  MoveL 690 to (-312.65, 5.37, -312.58) mm, rotated rx -179.15 ry 0 rz -30.08 deg; joints [-2.468, -65.05, 119.495, -183.449, 54.303, 242.138]
  MoveL 691 to (-312.62, 5.43, -312.23) mm, rotated rx -179.15 ry 0 rz -30.08 deg; joints [-2.467, -65.071, 119.523, -183.448, 54.309, 242.137]
  MoveL 692 to (-312.59, 5.47, -311.88) mm, rotated rx -179.15 ry 0 rz -30.08 deg; joints [-2.466, -65.091, 119.551, -183.447, 54.317, 242.136]
  MoveL 693 to (-312.58, 5.49, -311.54) mm, rotated rx -179.15 ry 0 rz -30.08 deg; joints [-2.466, -65.11, 119.579, -183.447, 54.326, 242.135]
  MoveL 694 to (-312.58, 5.49, -311.19) mm, rotated rx -179.15 ry 0 rz -30.08 deg; joints [-2.467, -65.129, 119.607, -183.447, 54.336, 242.135]
  MoveL 695 to (-312.58, 5.49, -5.24) mm, rotated rx -179.15 ry 0 rz -30.08 deg; joints [-3.196, -81.654, 142.775, -184.036, 60.99, 242.081]
  MoveL 696 to (-312.58, 5.49, -2.45) mm, rotated rx -179.15 ry 0 rz -30.08 deg; joints [-3.205, -81.818, 142.973, -184.044, 61.024, 242.083]
  MoveL 697 to (-312.59, 5.47, -2.1) mm, rotated rx -179.15 ry 0 rz -30.08 deg; joints [-3.206, -81.837, 142.998, -184.046, 61.03, 242.083]
  MoveL 698 to (-312.62, 5.43, -1.75) mm, rotated rx -179.15 ry 0 rz -30.08 deg; joints [-3.209, -81.854, 143.023, -184.049, 61.038, 242.084]
  MoveL 699 to (-312.65, 5.37, -1.4) mm, rotated rx -179.15 ry 0 rz -30.08 deg; joints [-3.212, -81.871, 143.049, -184.052, 61.048, 242.085]
  MoveL 700 to (-312.69, 5.3, -1.05) mm, rotated rx -179.15 ry 0 rz -30.08 deg; joints [-3.215, -81.886, 143.075, -184.055, 61.059, 242.086]
  MoveL 701 to (-312.75, 5.2, -0.7) mm, rotated rx -179.15 ry 0 rz -30.08 deg; joints [-3.22, -81.9, 143.102, -184.06, 61.072, 242.087]
  MoveL 702 to (-312.81, 5.09, -0.35) mm, rotated rx -179.15 ry 0 rz -30.08 deg; joints [-3.224, -81.912, 143.129, -184.065, 61.087, 242.089]
  MoveL 703 to (-312.89, 4.96, 0) mm, rotated rx -179.15 ry 0 rz -30.08 deg; joints [-3.23, -81.923, 143.156, -184.07, 61.103, 242.09]
  MoveL 704 to (-312.98, 4.8, 0.35) mm, rotated rx -179.15 ry 0 rz -30.08 deg; joints [-3.236, -81.932, 143.184, -184.077, 61.122, 242.092]
  MoveL 705 to (-313.06, 4.67, 0.61) mm, rotated rx -179.15 ry 0 rz -30.08 deg; joints [-3.242, -81.938, 143.205, -184.082, 61.138, 242.094]
  MoveL 706 to (-313.14, 4.52, 0.87) mm, rotated rx -179.15 ry 0 rz -30.08 deg; joints [-3.247, -81.942, 143.227, -184.088, 61.155, 242.096]
  MoveL 707 to (-313.28, 4.28, 1.23) mm, rotated rx -179.15 ry 0 rz -30.08 deg; joints [-3.256, -81.946, 143.257, -184.097, 61.181, 242.099]
  MoveL 708 to (-313.44, 4.01, 1.6) mm, rotated rx -179.15 ry 0 rz -30.08 deg; joints [-3.267, -81.948, 143.288, -184.108, 61.211, 242.102]
  MoveL 709 to (-313.54, 3.84, 1.8) mm, rotated rx -179.15 ry 0 rz -30.08 deg; joints [-3.273, -81.947, 143.306, -184.115, 61.23, 242.104]
  MoveL 710 to (-313.64, 3.66, 1.99) mm, rotated rx -179.15 ry 0 rz -30.08 deg; joints [-3.279, -81.945, 143.323, -184.121, 61.249, 242.106]
  MoveL 711 to (-313.84, 3.31, 2.32) mm, rotated rx -179.15 ry 0 rz -30.08 deg; joints [-3.292, -81.939, 143.354, -184.134, 61.286, 242.11]
  MoveL 712 to (-314.02, 3.01, 2.57) mm, rotated rx -179.15 ry 0 rz -30.08 deg; joints [-3.303, -81.932, 143.377, -184.145, 61.317, 242.113]
  MoveL 713 to (-314.19, 2.71, 2.78) mm, rotated rx -179.15 ry 0 rz -30.08 deg; joints [-3.314, -81.922, 143.398, -184.156, 61.348, 242.116]
  MoveL 714 to (-314.37, 2.41, 2.96) mm, rotated rx -179.15 ry 0 rz -30.08 deg; joints [-3.325, -81.91, 143.417, -184.167, 61.379, 242.12]
  MoveL 715 to (-314.54, 2.1, 3.12) mm, rotated rx -179.15 ry 0 rz -30.08 deg; joints [-3.335, -81.898, 143.435, -184.178, 61.41, 242.123]
  MoveL 716 to (-314.57, 2.06, 3.14) mm, rotated rx -179.15 ry 0 rz -30.08 deg; joints [-3.337, -81.896, 143.437, -184.18, 61.414, 242.123]
  MoveL 717 to (-314.74, 1.76, 3.27) mm, rotated rx -179.15 ry 0 rz -30.08 deg; joints [-3.347, -81.881, 143.452, -184.19, 61.443, 242.126]
  MoveL 718 to (-314.91, 1.47, 3.37) mm, rotated rx -179.15 ry 0 rz -30.08 deg; joints [-3.357, -81.866, 143.465, -184.201, 61.473, 242.129]
  MoveL 719 to (-315.08, 1.17, 3.46) mm, rotated rx -179.15 ry 0 rz -30.08 deg; joints [-3.367, -81.849, 143.477, -184.211, 61.502, 242.133]
  MoveL 720 to (-315.25, 0.88, 3.52) mm, rotated rx -179.15 ry 0 rz -30.08 deg; joints [-3.377, -81.831, 143.487, -184.222, 61.531, 242.136]
  MoveL 721 to (-315.43, 0.58, 3.57) mm, rotated rx -179.15 ry 0 rz -30.08 deg; joints [-3.387, -81.811, 143.497, -184.232, 61.559, 242.139]
  MoveL 722 to (-315.6, 0.28, 3.6) mm, rotated rx -179.15 ry 0 rz -30.08 deg; joints [-3.397, -81.791, 143.504, -184.242, 61.588, 242.142]
  MoveL 723 to (-315.94, -0.31, 3.61) mm, rotated rx -179.15 ry 0 rz -30.08 deg; joints [-3.417, -81.748, 143.517, -184.262, 61.644, 242.148]
  MoveL 724 to (-316.64, -1.52, 3.61) mm, rotated rx -179.15 ry 0 rz -30.08 deg; joints [-3.458, -81.658, 143.54, -184.304, 61.758, 242.16]
  MoveL 725 to (-316.99, -2.12, 3.58) mm, rotated rx -179.15 ry 0 rz -30.08 deg; joints [-3.478, -81.612, 143.551, -184.324, 61.815, 242.165]
  MoveL 726 to (-317.34, -2.72, 3.49) mm, rotated rx -179.15 ry 0 rz -30.08 deg; joints [-3.498, -81.562, 143.556, -184.344, 61.871, 242.171]
  MoveL 727 to (-321.53, -9.97, 2.16) mm, rotated rx -179.15 ry 0 rz -30.08 deg; joints [-3.734, -80.943, 143.599, -184.585, 62.54, 242.237]
  MoveL 728 to (-322.93, -12.38, 1.71) mm, rotated rx -179.15 ry 0 rz -30.08 deg; joints [-3.813, -80.735, 143.611, -184.664, 62.762, 242.257]
  MoveL 729 to (-323.1, -12.68, 1.62) mm, rotated rx -179.15 ry 0 rz -30.08 deg; joints [-3.823, -80.707, 143.61, -184.674, 62.788, 242.26]
  MoveL 730 to (-323.28, -12.97, 1.52) mm, rotated rx -179.15 ry 0 rz -30.08 deg; joints [-3.832, -80.679, 143.608, -184.683, 62.815, 242.262]
  MoveL 731 to (-323.45, -13.27, 1.39) mm, rotated rx -179.15 ry 0 rz -30.08 deg; joints [-3.841, -80.649, 143.604, -184.693, 62.841, 242.265]
  MoveL 732 to (-323.62, -13.56, 1.24) mm, rotated rx -179.15 ry 0 rz -30.08 deg; joints [-3.851, -80.618, 143.598, -184.702, 62.867, 242.267]
  MoveL 733 to (-323.79, -13.86, 1.06) mm, rotated rx -179.15 ry 0 rz -30.08 deg; joints [-3.86, -80.586, 143.591, -184.711, 62.892, 242.269]
  MoveL 734 to (-323.96, -14.15, 0.85) mm, rotated rx -179.15 ry 0 rz -30.08 deg; joints [-3.869, -80.552, 143.582, -184.72, 62.917, 242.272]
  MoveL 735 to (-324.13, -14.45, 0.62) mm, rotated rx -179.15 ry 0 rz -30.08 deg; joints [-3.878, -80.516, 143.57, -184.729, 62.942, 242.274]
  MoveL 736 to (-324.3, -14.74, 0.35) mm, rotated rx -179.15 ry 0 rz -30.08 deg; joints [-3.887, -80.478, 143.556, -184.738, 62.966, 242.276]
  MoveL 737 to (-324.33, -14.8, 0.3) mm, rotated rx -179.15 ry 0 rz -30.08 deg; joints [-3.888, -80.472, 143.554, -184.74, 62.97, 242.277]
  MoveC 738 to (-325.22, -16.33, 0.41) mm, rotated rx -179.15 ry 0 rz -30.08 deg; joints [-3.94, -80.362, 143.589, -184.791, 63.116, 242.289] to (-325.18, -16.27, 2.18) mm, rotated rx -179.15 ry 0 rz -30.08 deg; joints [-3.944, -80.467, 143.714, -184.796, 63.136, 242.29]
  MoveL 739 to (-325.18, -16.27, 2.18) mm, rotated rx -179.15 ry 0 rz -30.08 deg; joints [-3.944, -80.467, 143.714, -184.796, 63.136, 242.29]
  MoveL 740 to (-324.74, -15.51, 3.02) mm, rotated rx -179.15 ry 0 rz -30.08 deg; joints [-3.922, -80.573, 143.76, -184.774, 63.076, 242.284]
  Set speed (50.0 mm/s)
  MoveL 741 to (-322.97, -16.53, 3.02) mm, rotated rx -179.15 ry 0 rz -30.08 deg; joints [-3.82, -80.504, 143.789, -184.655, 63.169, 242.224]
  MoveL 742 to (-321.44, -16.41, 2.09) mm, rotated rx -179.15 ry 0 rz -30.08 deg; joints [-3.727, -80.466, 143.728, -184.552, 63.143, 242.179]
  Set speed (100.0 mm/s)
  MoveC 743 to (-321.26, -16.11, 1.18) mm, rotated rx -179.15 ry 0 rz -30.08 deg; joints [-3.714, -80.437, 143.658, -184.539, 63.101, 242.176] to (-321.46, -16.46, 0.3) mm, rotated rx -179.15 ry 0 rz -30.08 deg; joints [-3.722, -80.361, 143.601, -184.547, 63.121, 242.179]
  MoveL 744 to (-321.46, -16.46, 0.3) mm, rotated rx -179.15 ry 0 rz -30.08 deg; joints [-3.722, -80.361, 143.601, -184.547, 63.121, 242.179]
  MoveL 745 to (-321.65, -16.77, -0.05) mm, rotated rx -179.15 ry 0 rz -30.08 deg; joints [-3.732, -80.317, 143.582, -184.557, 63.146, 242.181]
  MoveL 746 to (-321.8, -17.04, -0.39) mm, rotated rx -179.15 ry 0 rz -30.08 deg; joints [-3.739, -80.277, 143.562, -184.565, 63.166, 242.183]
  MoveL 747 to (-321.94, -17.28, -0.73) mm, rotated rx -179.15 ry 0 rz -30.08 deg; joints [-3.746, -80.24, 143.542, -184.571, 63.183, 242.185]
  MoveL 748 to (-322.05, -17.48, -1.07) mm, rotated rx -179.15 ry 0 rz -30.08 deg; joints [-3.751, -80.205, 143.521, -184.577, 63.198, 242.186]
  MoveL 749 to (-322.16, -17.66, -1.42) mm, rotated rx -179.15 ry 0 rz -30.08 deg; joints [-3.756, -80.173, 143.5, -184.581, 63.209, 242.188]
  MoveL 750 to (-322.25, -17.81, -1.76) mm, rotated rx -179.15 ry 0 rz -30.08 deg; joints [-3.76, -80.142, 143.478, -184.585, 63.218, 242.189]
  MoveL 751 to (-322.32, -17.94, -2.1) mm, rotated rx -179.15 ry 0 rz -30.08 deg; joints [-3.763, -80.112, 143.456, -184.589, 63.226, 242.19]
  MoveL 752 to (-322.38, -18.05, -2.45) mm, rotated rx -179.15 ry 0 rz -30.08 deg; joints [-3.765, -80.085, 143.433, -184.591, 63.231, 242.19]
  MoveL 753 to (-322.44, -18.14, -2.8) mm, rotated rx -179.15 ry 0 rz -30.08 deg; joints [-3.767, -80.058, 143.41, -184.593, 63.235, 242.191]
  MoveL 754 to (-322.48, -18.22, -3.14) mm, rotated rx -179.15 ry 0 rz -30.08 deg; joints [-3.768, -80.033, 143.386, -184.594, 63.236, 242.191]
  MoveL 755 to (-322.51, -18.27, -3.49) mm, rotated rx -179.15 ry 0 rz -30.08 deg; joints [-3.769, -80.009, 143.362, -184.595, 63.236, 242.192]
  MoveL 756 to (-322.54, -18.31, -3.84) mm, rotated rx -179.15 ry 0 rz -30.08 deg; joints [-3.769, -79.986, 143.338, -184.595, 63.235, 242.192]
  MoveL 757 to (-322.55, -18.33, -4.19) mm, rotated rx -179.15 ry 0 rz -30.08 deg; joints [-3.768, -79.964, 143.314, -184.594, 63.232, 242.192]
  MoveL 758 to (-322.55, -18.34, -4.54) mm, rotated rx -179.15 ry 0 rz -30.08 deg; joints [-3.767, -79.944, 143.289, -184.593, 63.227, 242.192]
  MoveL 759 to (-322.55, -18.34, -311.19) mm, rotated rx -179.15 ry 0 rz -30.08 deg; joints [-2.902, -63.912, 119.964, -183.907, 55.922, 242.314]
  MoveL 760 to (-322.55, -18.33, -311.54) mm, rotated rx -179.15 ry 0 rz -30.08 deg; joints [-2.901, -63.895, 119.935, -183.906, 55.911, 242.314]
  MoveL 761 to (-322.54, -18.31, -311.88) mm, rotated rx -179.15 ry 0 rz -30.08 deg; joints [-2.9, -63.878, 119.906, -183.905, 55.898, 242.314]
  MoveL 762 to (-322.51, -18.27, -312.23) mm, rotated rx -179.15 ry 0 rz -30.08 deg; joints [-2.898, -63.863, 119.877, -183.904, 55.885, 242.314]
  MoveL 763 to (-322.48, -18.22, -312.58) mm, rotated rx -179.15 ry 0 rz -30.08 deg; joints [-2.896, -63.848, 119.848, -183.902, 55.87, 242.314]
  MoveL 764 to (-322.44, -18.14, -312.93) mm, rotated rx -179.15 ry 0 rz -30.08 deg; joints [-2.894, -63.834, 119.818, -183.899, 55.854, 242.313]
  MoveL 765 to (-322.38, -18.05, -313.28) mm, rotated rx -179.15 ry 0 rz -30.08 deg; joints [-2.89, -63.821, 119.789, -183.896, 55.837, 242.312]
  MoveL 766 to (-322.32, -17.93, -313.63) mm, rotated rx -179.15 ry 0 rz -30.08 deg; joints [-2.887, -63.81, 119.759, -183.893, 55.819, 242.311]
  MoveL 767 to (-322.24, -17.8, -313.98) mm, rotated rx -179.15 ry 0 rz -30.08 deg; joints [-2.883, -63.799, 119.728, -183.889, 55.799, 242.31]
  MoveL 768 to (-322.15, -17.64, -314.33) mm, rotated rx -179.15 ry 0 rz -30.08 deg; joints [-2.878, -63.789, 119.698, -183.884, 55.778, 242.309]
  MoveL 769 to (-322.05, -17.46, -314.68) mm, rotated rx -179.15 ry 0 rz -30.08 deg; joints [-2.873, -63.781, 119.667, -183.879, 55.755, 242.307]
  MoveL 770 to (-321.92, -17.25, -315.03) mm, rotated rx -179.15 ry 0 rz -30.08 deg; joints [-2.867, -63.774, 119.635, -183.873, 55.73, 242.305]
  MoveL 771 to (-321.78, -17.01, -315.38) mm, rotated rx -179.15 ry 0 rz -30.08 deg; joints [-2.86, -63.769, 119.603, -183.866, 55.703, 242.303]
  MoveL 772 to (-321.63, -16.75, -315.7) mm, rotated rx -179.15 ry 0 rz -30.08 deg; joints [-2.853, -63.766, 119.574, -183.858, 55.676, 242.3]
  MoveL 773 to (-321.46, -16.46, -316.02) mm, rotated rx -179.15 ry 0 rz -30.08 deg; joints [-2.844, -63.765, 119.543, -183.85, 55.647, 242.297]
  MoveL 774 to (-321.29, -16.16, -316.3) mm, rotated rx -179.15 ry 0 rz -30.08 deg; joints [-2.836, -63.767, 119.516, -183.841, 55.618, 242.293]
  MoveL 775 to (-321.11, -15.85, -316.55) mm, rotated rx -179.15 ry 0 rz -30.08 deg; joints [-2.828, -63.77, 119.492, -183.832, 55.591, 242.29]
  MoveL 776 to (-320.94, -15.55, -316.76) mm, rotated rx -179.15 ry 0 rz -30.08 deg; joints [-2.82, -63.775, 119.471, -183.824, 55.564, 242.287]
  MoveL 777 to (-320.76, -15.25, -316.94) mm, rotated rx -179.15 ry 0 rz -30.08 deg; joints [-2.812, -63.781, 119.452, -183.815, 55.538, 242.283]
  MoveL 778 to (-320.59, -14.95, -317.1) mm, rotated rx -179.15 ry 0 rz -30.08 deg; joints [-2.804, -63.789, 119.435, -183.807, 55.514, 242.28]
  MoveL 779 to (-320.41, -14.65, -317.23) mm, rotated rx -179.15 ry 0 rz -30.08 deg; joints [-2.796, -63.798, 119.42, -183.798, 55.489, 242.276]
  MoveL 780 to (-320.24, -14.35, -317.34) mm, rotated rx -179.15 ry 0 rz -30.08 deg; joints [-2.788, -63.808, 119.407, -183.79, 55.466, 242.273]
  MoveL 781 to (-320.06, -14.04, -317.43) mm, rotated rx -179.15 ry 0 rz -30.08 deg; joints [-2.781, -63.819, 119.395, -183.781, 55.443, 242.269]
  MoveL 782 to (-319.89, -13.74, -317.5) mm, rotated rx -179.15 ry 0 rz -30.08 deg; joints [-2.773, -63.831, 119.386, -183.773, 55.421, 242.266]
  MoveL 783 to (-319.71, -13.44, -317.55) mm, rotated rx -179.15 ry 0 rz -30.08 deg; joints [-2.765, -63.844, 119.378, -183.765, 55.4, 242.262]
  MoveL 784 to (-319.54, -13.14, -317.58) mm, rotated rx -179.15 ry 0 rz -30.08 deg; joints [-2.758, -63.858, 119.371, -183.756, 55.379, 242.259]
  MoveL 785 to (-319.37, -12.84, -317.59) mm, rotated rx -179.15 ry 0 rz -30.08 deg; joints [-2.75, -63.873, 119.366, -183.748, 55.359, 242.255]
  MoveL 786 to (-312.02, -0.16, -317.59) mm, rotated rx -179.15 ry 0 rz -30.08 deg; joints [-2.43, -64.521, 119.184, -183.394, 54.519, 242.095]
  MoveL 787 to (-311.85, 0.14, -317.58) mm, rotated rx -179.15 ry 0 rz -30.08 deg; joints [-2.423, -64.536, 119.18, -183.385, 54.499, 242.091]
  MoveL 788 to (-311.67, 0.44, -317.56) mm, rotated rx -179.15 ry 0 rz -30.08 deg; joints [-2.415, -64.552, 119.177, -183.377, 54.48, 242.087]
  MoveL 789 to (-311.5, 0.74, -317.53) mm, rotated rx -179.15 ry 0 rz -30.08 deg; joints [-2.408, -64.57, 119.175, -183.368, 54.461, 242.083]
  MoveL 790 to (-311.32, 1.05, -317.47) mm, rotated rx -179.15 ry 0 rz -30.08 deg; joints [-2.4, -64.588, 119.175, -183.36, 54.443, 242.079]
  MoveL 791 to (-311.15, 1.35, -317.39) mm, rotated rx -179.15 ry 0 rz -30.08 deg; joints [-2.393, -64.607, 119.177, -183.352, 54.425, 242.075]
  MoveL 792 to (-310.97, 1.65, -317.29) mm, rotated rx -179.15 ry 0 rz -30.08 deg; joints [-2.385, -64.627, 119.181, -183.343, 54.408, 242.071]
  MoveL 793 to (-310.8, 1.95, -317.17) mm, rotated rx -179.15 ry 0 rz -30.08 deg; joints [-2.378, -64.649, 119.186, -183.335, 54.392, 242.067]
  MoveL 794 to (-310.62, 2.25, -317.03) mm, rotated rx -179.15 ry 0 rz -30.08 deg; joints [-2.37, -64.672, 119.193, -183.326, 54.376, 242.063]
  MoveL 795 to (-310.45, 2.55, -316.86) mm, rotated rx -179.15 ry 0 rz -30.08 deg; joints [-2.363, -64.696, 119.202, -183.318, 54.361, 242.059]
  MoveL 796 to (-310.28, 2.86, -316.66) mm, rotated rx -179.15 ry 0 rz -30.08 deg; joints [-2.356, -64.721, 119.214, -183.31, 54.347, 242.054]
  MoveL 797 to (-310.09, 3.18, -316.41) mm, rotated rx -179.15 ry 0 rz -30.08 deg; joints [-2.348, -64.75, 119.229, -183.3, 54.332, 242.05]
  MoveL 798 to (-309.9, 3.51, -316.12) mm, rotated rx -179.15 ry 0 rz -30.08 deg; joints [-2.34, -64.782, 119.248, -183.291, 54.319, 242.045]
  MoveL 799 to (-309.71, 3.84, -315.78) mm, rotated rx -179.15 ry 0 rz -30.08 deg; joints [-2.333, -64.816, 119.27, -183.282, 54.308, 242.04]
  MoveL 800 to (-309.52, 4.16, -315.38) mm, rotated rx -179.15 ry 0 rz -30.08 deg; joints [-2.325, -64.853, 119.298, -183.274, 54.298, 242.036]
  MoveL 801 to (-309.4, 4.37, -315.08) mm, rotated rx -179.15 ry 0 rz -30.08 deg; joints [-2.32, -64.879, 119.319, -183.268, 54.293, 242.033]
  MoveL 802 to (-309.29, 4.55, -314.79) mm, rotated rx -179.15 ry 0 rz -30.08 deg; joints [-2.316, -64.903, 119.34, -183.263, 54.29, 242.03]
  MoveL 803 to (-309.2, 4.71, -314.5) mm, rotated rx -179.15 ry 0 rz -30.08 deg; joints [-2.313, -64.927, 119.362, -183.259, 54.288, 242.028]
  MoveL 804 to (-309.12, 4.86, -314.2) mm, rotated rx -179.15 ry 0 rz -30.08 deg; joints [-2.309, -64.949, 119.383, -183.255, 54.287, 242.025]
  MoveL 805 to (-309.04, 4.98, -313.91) mm, rotated rx -179.15 ry 0 rz -30.08 deg; joints [-2.307, -64.971, 119.405, -183.252, 54.287, 242.023]
  MoveL 806 to (-308.98, 5.09, -313.62) mm, rotated rx -179.15 ry 0 rz -30.08 deg; joints [-2.304, -64.991, 119.428, -183.249, 54.289, 242.022]
  MoveL 807 to (-308.88, 5.27, -313.03) mm, rotated rx -179.15 ry 0 rz -30.08 deg; joints [-2.301, -65.031, 119.473, -183.244, 54.294, 242.019]
  MoveL 808 to (-308.82, 5.37, -312.58) mm, rotated rx -179.15 ry 0 rz -30.08 deg; joints [-2.299, -65.059, 119.507, -183.242, 54.301, 242.017]
  MoveL 809 to (-308.79, 5.43, -312.23) mm, rotated rx -179.15 ry 0 rz -30.08 deg; joints [-2.298, -65.08, 119.535, -183.24, 54.307, 242.016]
  MoveL 810 to (-308.76, 5.47, -311.88) mm, rotated rx -179.15 ry 0 rz -30.08 deg; joints [-2.298, -65.1, 119.563, -183.24, 54.315, 242.015]
  MoveL 811 to (-308.75, 5.49, -311.54) mm, rotated rx -179.15 ry 0 rz -30.08 deg; joints [-2.298, -65.119, 119.591, -183.239, 54.324, 242.015]
  MoveL 812 to (-308.75, 5.49, -311.19) mm, rotated rx -179.15 ry 0 rz -30.08 deg; joints [-2.298, -65.137, 119.619, -183.239, 54.334, 242.014]
  MoveL 813 to (-308.75, 5.49, -5.24) mm, rotated rx -179.15 ry 0 rz -30.08 deg; joints [-2.976, -81.666, 142.789, -183.784, 60.984, 241.959]
  MoveL 814 to (-308.75, 5.49, -2.45) mm, rotated rx -179.15 ry 0 rz -30.08 deg; joints [-2.984, -81.83, 142.987, -183.792, 61.018, 241.961]
  MoveL 815 to (-308.76, 5.46, -2.07) mm, rotated rx -179.15 ry 0 rz -30.08 deg; joints [-2.986, -81.85, 143.014, -183.794, 61.025, 241.962]
  MoveL 816 to (-308.79, 5.42, -1.7) mm, rotated rx -179.15 ry 0 rz -30.08 deg; joints [-2.988, -81.869, 143.041, -183.797, 61.034, 241.963]
  MoveL 817 to (-308.83, 5.36, -1.32) mm, rotated rx -179.15 ry 0 rz -30.08 deg; joints [-2.992, -81.887, 143.069, -183.8, 61.044, 241.964]
  MoveL 818 to (-308.88, 5.27, -0.95) mm, rotated rx -179.15 ry 0 rz -30.08 deg; joints [-2.996, -81.902, 143.097, -183.804, 61.056, 241.965]
  MoveL 819 to (-308.93, 5.18, -0.63) mm, rotated rx -179.15 ry 0 rz -30.08 deg; joints [-3, -81.915, 143.122, -183.808, 61.069, 241.966]
  MoveL 820 to (-308.99, 5.07, -0.3) mm, rotated rx -179.15 ry 0 rz -30.08 deg; joints [-3.004, -81.926, 143.147, -183.813, 61.083, 241.968]
  MoveL 821 to (-309.06, 4.95, 0.02) mm, rotated rx -179.15 ry 0 rz -30.08 deg; joints [-3.009, -81.936, 143.172, -183.818, 61.099, 241.969]
  MoveL 822 to (-309.15, 4.8, 0.35) mm, rotated rx -179.15 ry 0 rz -30.08 deg; joints [-3.015, -81.945, 143.198, -183.824, 61.116, 241.971]
  MoveL 823 to (-309.24, 4.65, 0.64) mm, rotated rx -179.15 ry 0 rz -30.08 deg; joints [-3.021, -81.951, 143.222, -183.83, 61.134, 241.973]
  MoveL 824 to (-309.33, 4.48, 0.93) mm, rotated rx -179.15 ry 0 rz -30.08 deg; joints [-3.027, -81.956, 143.246, -183.837, 61.153, 241.975]
  MoveL 825 to (-309.44, 4.29, 1.22) mm, rotated rx -179.15 ry 0 rz -30.08 deg; joints [-3.035, -81.959, 143.271, -183.844, 61.174, 241.977]
  MoveL 826 to (-309.57, 4.08, 1.51) mm, rotated rx -179.15 ry 0 rz -30.08 deg; joints [-3.043, -81.961, 143.295, -183.853, 61.198, 241.98]
  MoveL 827 to (-309.75, 3.77, 1.87) mm, rotated rx -179.15 ry 0 rz -30.08 deg; joints [-3.054, -81.96, 143.327, -183.864, 61.231, 241.983]
  MoveL 828 to (-309.92, 3.47, 2.18) mm, rotated rx -179.15 ry 0 rz -30.08 deg; joints [-3.065, -81.955, 143.355, -183.876, 61.264, 241.987]
  MoveL 829 to (-310.1, 3.16, 2.45) mm, rotated rx -179.15 ry 0 rz -30.08 deg; joints [-3.076, -81.949, 143.38, -183.887, 61.296, 241.991]
  MoveL 830 to (-310.28, 2.86, 2.68) mm, rotated rx -179.15 ry 0 rz -30.08 deg; joints [-3.087, -81.94, 143.403, -183.898, 61.327, 241.994]
  MoveL 831 to (-310.39, 2.66, 2.81) mm, rotated rx -179.15 ry 0 rz -30.08 deg; joints [-3.094, -81.933, 143.416, -183.906, 61.347, 241.996]
  MoveL 832 to (-310.51, 2.46, 2.93) mm, rotated rx -179.15 ry 0 rz -30.08 deg; joints [-3.101, -81.926, 143.429, -183.913, 61.368, 241.999]
  MoveL 833 to (-310.74, 2.06, 3.14) mm, rotated rx -179.15 ry 0 rz -30.08 deg; joints [-3.115, -81.909, 143.451, -183.927, 61.408, 242.003]
  MoveL 834 to (-310.97, 1.66, 3.31) mm, rotated rx -179.15 ry 0 rz -30.08 deg; joints [-3.129, -81.889, 143.471, -183.942, 61.448, 242.007]
  MoveL 835 to (-311.2, 1.25, 3.44) mm, rotated rx -179.15 ry 0 rz -30.08 deg; joints [-3.143, -81.866, 143.489, -183.956, 61.488, 242.012]
  MoveL 836 to (-311.44, 0.85, 3.53) mm, rotated rx -179.15 ry 0 rz -30.08 deg; joints [-3.156, -81.842, 143.503, -183.97, 61.527, 242.016]
  MoveL 837 to (-311.67, 0.44, 3.59) mm, rotated rx -179.15 ry 0 rz -30.08 deg; joints [-3.17, -81.815, 143.515, -183.984, 61.566, 242.021]
  MoveL 838 to (-311.85, 0.14, 3.6) mm, rotated rx -179.15 ry 0 rz -30.08 deg; joints [-3.18, -81.794, 143.523, -183.995, 61.595, 242.024]
  MoveL 839 to (-312.02, -0.16, 3.61) mm, rotated rx -179.15 ry 0 rz -30.08 deg; joints [-3.19, -81.772, 143.529, -184.005, 61.624, 242.027]
  MoveL 840 to (-313.77, -3.18, 3.61) mm, rotated rx -179.15 ry 0 rz -30.08 deg; joints [-3.291, -81.548, 143.588, -184.109, 61.91, 242.058]
  MoveL 841 to (-314.12, -3.78, 3.58) mm, rotated rx -179.15 ry 0 rz -30.08 deg; joints [-3.311, -81.502, 143.598, -184.129, 61.967, 242.064]
  MoveL 842 to (-314.47, -4.39, 3.49) mm, rotated rx -179.15 ry 0 rz -30.08 deg; joints [-3.331, -81.452, 143.603, -184.15, 62.023, 242.07]
  MoveL 843 to (-318.67, -11.63, 2.16) mm, rotated rx -179.15 ry 0 rz -30.08 deg; joints [-3.568, -80.832, 143.646, -184.391, 62.691, 242.138]
  MoveL 844 to (-320.06, -14.04, 1.71) mm, rotated rx -179.15 ry 0 rz -30.08 deg; joints [-3.647, -80.624, 143.658, -184.471, 62.913, 242.159]
  MoveL 845 to (-320.24, -14.34, 1.62) mm, rotated rx -179.15 ry 0 rz -30.08 deg; joints [-3.657, -80.597, 143.657, -184.481, 62.94, 242.161]
  MoveL 846 to (-320.41, -14.63, 1.52) mm, rotated rx -179.15 ry 0 rz -30.08 deg; joints [-3.666, -80.568, 143.655, -184.49, 62.966, 242.164]
  MoveL 847 to (-320.58, -14.93, 1.39) mm, rotated rx -179.15 ry 0 rz -30.08 deg; joints [-3.676, -80.538, 143.651, -184.5, 62.992, 242.166]
  MoveL 848 to (-320.75, -15.22, 1.24) mm, rotated rx -179.15 ry 0 rz -30.08 deg; joints [-3.685, -80.507, 143.645, -184.509, 63.018, 242.169]
  MoveL 849 to (-320.92, -15.52, 1.06) mm, rotated rx -179.15 ry 0 rz -30.08 deg; joints [-3.694, -80.475, 143.638, -184.519, 63.044, 242.171]
  MoveL 850 to (-321.09, -15.82, 0.85) mm, rotated rx -179.15 ry 0 rz -30.08 deg; joints [-3.703, -80.441, 143.629, -184.528, 63.069, 242.174]
  MoveL 851 to (-321.26, -16.11, 0.62) mm, rotated rx -179.15 ry 0 rz -30.08 deg; joints [-3.712, -80.405, 143.617, -184.537, 63.093, 242.176]
  MoveL 852 to (-321.43, -16.41, 0.35) mm, rotated rx -179.15 ry 0 rz -30.08 deg; joints [-3.721, -80.367, 143.603, -184.546, 63.117, 242.178]
  MoveL 853 to (-321.46, -16.46, 0.3) mm, rotated rx -179.15 ry 0 rz -30.08 deg; joints [-3.722, -80.361, 143.601, -184.547, 63.121, 242.179]
  MoveC 854 to (-321.99, -17.38, 0.01) mm, rotated rx -179.15 ry 0 rz -30.08 deg; joints [-3.752, -80.275, 143.596, -184.577, 63.204, 242.186] to (-322.44, -18.14, 0.66) mm, rotated rx -179.15 ry 0 rz -30.08 deg; joints [-3.78, -80.253, 143.656, -184.605, 63.286, 242.193]
  MoveL 855 to (-322.44, -18.14, 0.66) mm, rotated rx -179.15 ry 0 rz -30.08 deg; joints [-3.78, -80.253, 143.656, -184.605, 63.286, 242.193]
  MoveL 856 to (-323.43, -19.85, 4.32) mm, rotated rx -179.15 ry 0 rz -30.08 deg; joints [-3.85, -80.331, 143.946, -184.675, 63.5, 242.209]
  MoveL 857 to (-324.83, -19.73, 5.44) mm, rotated rx -179.15 ry 0 rz -30.08 deg; joints [-3.936, -80.397, 144.017, -184.771, 63.508, 242.251]
  Set speed (200.0 mm/s)
  MoveL 858 to (-336.31, -13.08, 5.44) mm, rotated rx -179.15 ry 0 rz -30.08 deg; joints [-4.602, -80.84, 143.822, -185.545, 62.9, 242.649]
  Print: /'Parallel1'
  Call SetTool(1)
  Set speed (200.0 mm/s)
  MoveL 859 to (-340.11, 16.27, -316.36) mm, rotated rx -179.15 ry 0 rz -30.08 deg; joints [-3.663, -65.306, 118.877, -184.975, 53.482, 243.085]
  MoveL 860 to (-319.42, 4.29, -316.36) mm, rotated rx -179.15 ry 0 rz -30.08 deg; joints [-2.757, -64.785, 119.182, -183.807, 54.266, 242.348]
  Set speed (100.0 mm/s)
  MoveL 861 to (-318.78, 3.92, -316.36) mm, rotated rx -179.15 ry 0 rz -30.08 deg; joints [-2.729, -64.769, 119.191, -183.772, 54.289, 242.326]
  MoveC 862 to (-318.01, 3.47, -315.99) mm, rotated rx -179.15 ry 0 rz -30.08 deg; joints [-2.696, -64.768, 119.232, -183.729, 54.33, 242.299] to (-317.69, 3.28, -315.09) mm, rotated rx -179.15 ry 0 rz -30.08 deg; joints [-2.683, -64.806, 119.309, -183.712, 54.369, 242.287]
  MoveL 863 to (-317.69, 3.28, -315.09) mm, rotated rx -179.15 ry 0 rz -30.08 deg; joints [-2.683, -64.806, 119.309, -183.712, 54.369, 242.287]
  MoveL 864 to (-317.69, 3.28, 0.74) mm, rotated rx -179.15 ry 0 rz -30.08 deg; joints [-3.509, -81.83, 143.227, -184.382, 61.276, 242.229]
  MoveL 865 to (-317.74, 3.32, 1.02) mm, rotated rx -179.15 ry 0 rz -30.08 deg; joints [-3.513, -81.849, 143.246, -184.387, 61.276, 242.231]
  MoveL 866 to (-317.8, 3.35, 1.3) mm, rotated rx -179.15 ry 0 rz -30.08 deg; joints [-3.517, -81.867, 143.265, -184.392, 61.277, 242.234]
  MoveL 867 to (-317.8, 3.35, 2.99) mm, rotated rx -179.15 ry 0 rz -30.08 deg; joints [-3.523, -81.967, 143.384, -184.397, 61.297, 242.235]
  MoveC 868 to (-318.08, 2.86, 4.33) mm, rotated rx -179.15 ry 0 rz -30.08 deg; joints [-3.544, -82.011, 143.489, -184.419, 61.358, 242.241] to (-318.75, 1.7, 4.89) mm, rotated rx -179.15 ry 0 rz -30.08 deg; joints [-3.585, -81.957, 143.551, -184.46, 61.475, 242.253]
  MoveL 869 to (-318.75, 1.7, 4.89) mm, rotated rx -179.15 ry 0 rz -30.08 deg; joints [-3.585, -81.957, 143.551, -184.46, 61.475, 242.253]
  MoveL 870 to (-320.03, -0.5, 4.89) mm, rotated rx -179.15 ry 0 rz -30.08 deg; joints [-3.658, -81.794, 143.595, -184.535, 61.684, 242.274]
  MoveC 871 to (-320.7, -1.66, 4.33) mm, rotated rx -179.15 ry 0 rz -30.08 deg; joints [-3.695, -81.675, 143.578, -184.572, 61.788, 242.284] to (-320.98, -2.15, 2.99) mm, rotated rx -179.15 ry 0 rz -30.08 deg; joints [-3.707, -81.56, 143.492, -184.584, 61.817, 242.288]
  MoveL 872 to (-320.98, -2.15, 2.99) mm, rotated rx -179.15 ry 0 rz -30.08 deg; joints [-3.707, -81.56, 143.492, -184.584, 61.817, 242.288]
  MoveL 873 to (-320.92, -2.18, 2.71) mm, rotated rx -179.15 ry 0 rz -30.08 deg; joints [-3.702, -81.542, 143.473, -184.579, 61.816, 242.286]
  MoveL 874 to (-320.87, -2.21, 2.43) mm, rotated rx -179.15 ry 0 rz -30.08 deg; joints [-3.698, -81.523, 143.454, -184.574, 61.816, 242.283]
  MoveL 875 to (-320.87, -2.21, -317.02) mm, rotated rx -179.15 ry 0 rz -30.08 deg; joints [-2.818, -64.427, 119.233, -183.863, 54.676, 242.358]
  MoveL 876 to (-320.92, -2.18, -317.3) mm, rotated rx -179.15 ry 0 rz -30.08 deg; joints [-2.82, -64.414, 119.21, -183.866, 54.666, 242.36]
  MoveL 877 to (-320.98, -2.15, -317.58) mm, rotated rx -179.15 ry 0 rz -30.08 deg; joints [-2.822, -64.401, 119.186, -183.869, 54.655, 242.363]
  MoveL 878 to (-320.98, -2.15, -317.58) mm, rotated rx -179.15 ry 0 rz -30.08 deg; joints [-2.822, -64.401, 119.186, -183.869, 54.655, 242.363]
  MoveC 879 to (-321.26, -2.63, -318.92) mm, rotated rx -179.15 ry 0 rz -30.08 deg; joints [-2.831, -64.308, 119.083, -183.881, 54.646, 242.37] to (-321.94, -3.79, -319.48) mm, rotated rx -179.15 ry 0 rz -30.08 deg; joints [-2.859, -64.22, 119.054, -183.912, 54.706, 242.385]
  MoveL 880 to (-321.94, -3.79, -319.48) mm, rotated rx -179.15 ry 0 rz -30.08 deg; joints [-2.859, -64.22, 119.054, -183.912, 54.706, 242.385]
  MoveL 881 to (-323.21, -5.99, -319.48) mm, rotated rx -179.15 ry 0 rz -30.08 deg; joints [-2.915, -64.108, 119.085, -183.973, 54.851, 242.412]
  MoveC 882 to (-323.88, -7.16, -318.92) mm, rotated rx -179.15 ry 0 rz -30.08 deg; joints [-2.945, -64.077, 119.148, -184.006, 54.945, 242.425] to (-324.16, -7.64, -317.58) mm, rotated rx -179.15 ry 0 rz -30.08 deg; joints [-2.96, -64.121, 119.265, -184.02, 55.019, 242.429]
  MoveL 883 to (-324.16, -7.64, -317.58) mm, rotated rx -179.15 ry 0 rz -30.08 deg; joints [-2.96, -64.121, 119.265, -184.02, 55.019, 242.429]
  MoveL 884 to (-324.11, -7.67, -317.3) mm, rotated rx -179.15 ry 0 rz -30.08 deg; joints [-2.959, -64.133, 119.288, -184.018, 55.029, 242.427]
  MoveL 885 to (-324.11, -7.67, -317.3) mm, rotated rx -179.15 ry 0 rz -30.08 deg; joints [-2.959, -64.134, 119.288, -184.018, 55.029, 242.427]
  MoveL 886 to (-324.05, -7.7, -317.02) mm, rotated rx -179.15 ry 0 rz -30.08 deg; joints [-2.957, -64.146, 119.312, -184.015, 55.04, 242.425]
  MoveL 887 to (-324.05, -7.7, 1.46) mm, rotated rx -179.15 ry 0 rz -30.08 deg; joints [-3.877, -81.057, 143.49, -184.756, 62.322, 242.332]
  MoveC 888 to (-324.37, -7.52, 2.36) mm, rotated rx -179.15 ry 0 rz -30.08 deg; joints [-3.899, -81.121, 143.548, -184.781, 62.317, 242.344] to (-325.15, -7.07, 2.73) mm, rotated rx -179.15 ry 0 rz -30.08 deg; joints [-3.946, -81.172, 143.561, -184.835, 62.281, 242.371]
  MoveL 889 to (-325.15, -7.07, 2.73) mm, rotated rx -179.15 ry 0 rz -30.08 deg; joints [-3.946, -81.172, 143.561, -184.835, 62.281, 242.371]
  Set speed (200.0 mm/s)
  MoveL 890 to (-346.48, 5.29, 2.73) mm, rotated rx -179.15 ry 0 rz -30.08 deg; joints [-5.178, -81.959, 143.173, -186.294, 61.169, 243.159]
  MoveL 891 to (-346.48, 5.29, 2.73) mm, rotated rx -179.15 ry 0 rz -30.08 deg; joints [-5.178, -81.959, 143.173, -186.294, 61.169, 243.159]
